FUNCTION_BLOCK MockAbortable EXTENDS Object IMPLEMENTS I_Abortable
VAR
	_isRegistered : BOOL;
END_VAR

METHOD Abort : Base_Library.HRESULT
END_METHOD

METHOD IsRegistered : BOOL
VAR_INPUT
END_VAR
IsRegistered := _isRegistered;
END_METHOD

METHOD RegisterWithParent
VAR_INPUT
	Parent	: I_HostObjects;
END_VAR
IF NOT _isRegistered THEN
	IF SUCCEEDED(Parent.RegisterAbortable(THIS^)) THEN
		_isRegistered := TRUE;
	ELSE
		_isRegistered := FALSE;
	END_IF
END_IF
END_METHOD

END_FUNCTION_BLOCK

(* stored: Version 1.1.0.1
   POU MockAbortable: Id {a3a08092-5752-4e7b-aa34-7940d1bedfee}, SpecialFunc None
   Method Abort: Id {a05f445d-bf80-4bb4-bca8-4dc23e0ac783}
   Method IsRegistered: Id {af0b5ed4-894f-4e18-8c38-e6f757d31458}
   Method RegisterWithParent: Id {06e7efa5-26d0-4737-a95a-25426fc72b67} *)
